// TIA Portal V17 export
// export: Created 2024-08-26T21:07:16.6253972Z, ExportSetting WithDefaults, DisplayName Totally Integrated Automation Portal, DisplayVersion V17 Update 7, DisplayName TIA Portal Openness, DisplayVersion V17 Update 7, DisplayName TIA Portal Version Control Interface, DisplayVersion V17, DisplayName SINAMICS Startdrive Advanced, DisplayVersion V17 SP2, DisplayName SINAMICS Startdrive G110M, G120, G120C, G120D, G120P, G115D, DisplayVersion V17 SP2, DisplayName SINAMICS Startdrive G130, G150, S120, S150, SINAMICS MV, S210, DisplayVersion V17 SP2, DisplayName STEP 7 Professional, DisplayVersion V17 Update 7, DisplayName STEP 7 Safety, DisplayVersion V17 Update 6, DisplayName WinCC Advanced / Unified PC, DisplayVersion V17 Update 7
DATA_BLOCK "torque"   // DB34
{ S7_Optimized_Access := 'TRUE' }
VERSION : 0.1
// stored: AutoNumber true, DBAccessibleFromOPCUA true, DBAccessibleFromWebserver true, IsOnlyStoredInLoadMemory false, IsRetainMemResEnabled false, IsWriteProtectedInAS false, MemoryReserve 100
   VAR
      ON : Bool := FALSE;
      SENSOR : Int := 0;
      TORQUE : Int := 0;
      TIMER1 { S7_SetPoint := 'True'} : TON_TIME;
      TIMER2 { S7_SetPoint := 'True'} : TON_TIME;
      TIMER3 { S7_SetPoint := 'True'} : TON_TIME;
      TIMER4 { S7_SetPoint := 'True'} : TON_TIME;
      TIMER5 { S7_SetPoint := 'True'} : TON_TIME;
      "1stInt" : Word := 16#0000;
      "2ndInt" : Word := 16#0000;
      "3rdInt" : Word := 16#0000;
      "4thInt" : Word := 16#0000;
      "5thInt" : Word := 16#0000;
      "1stDecimal" : Word := 16#0000;
      "2ndDecimal" : Word := 16#0000;
      "3rdDecimal" : Word := 16#0000;
      "4thDecimal" : Word := 16#0000;
      "5thDecimal" : Word := 16#0000;
      "1stFinalAngle" : Word := 16#0000;
      "2ndFinalAngle" : Word := 16#0000;
      "3rdFinalAngle" : Word := 16#0000;
      "4thFinalAngle" : Word := 16#0000;
      "5thFinalAngle" : Word := 16#0000;
      "ENTERO MANUAL" : Word := 16#0000;
      "DECIMAL MANUAL" : Word := 16#0000;
      "ANGULO FINAL MANUAL" : Word := 16#0000;
      TORNILLO : Int := 0;
      "1Ok" : Bool := FALSE;
      "2Ok" : Bool := FALSE;
      "3Ok" : Bool := FALSE;
      "4Ok" : Bool := FALSE;
      "1_OK_2" : Bool := FALSE;
      "2_OK_2" : Bool := FALSE;
      "3_OK_2" : Bool := FALSE;
      "4_OK_2" : Bool := FALSE;
      "5_OK_2" : Bool := FALSE;
      "5_OK" : Bool := FALSE;
      "ACTIVAR MANUAL" : Bool := FALSE;
      "CONFIG1 MANUAL" : Bool := FALSE;
      "CONFIG2 MANUAL" : Bool := FALSE;
      "CONFIG3 MANUAL" : Bool := FALSE;
      "CONFIG4 MANUAL" : Bool := FALSE;
      "CONFIG5 MANUAL" : Bool := FALSE;
      "REINICIAR PFJOB" : Bool := FALSE;
      PRESET1 : Int := 0;
      PRESET2 : Int := 0;
      PRESET3 : Int := 0;
      PRESET4 : Int := 0;
      PRESET5 : Int := 0;
      manual2 : Struct
         HABILITAR : Bool := TRUE;
         DESHABILITAR : Bool := FALSE;
         BORRAR : Bool := FALSE;
      END_STRUCT;
      BLOQUEO : Array[0..6] of Bool;
      manual : Struct
         activate : Bool := TRUE;
         deactivate : Bool := FALSE;
         erase : Bool := FALSE;
      END_STRUCT;
   END_VAR
   VAR RETAIN
      "P6000 TORQUE_1" : Array[0..15] of Int;
      p6000Torque : Array[0..15] of Int;
   END_VAR
   VAR
      nok2 : Array[0..1] of Bool;
      nok : Array[0..1] of Bool;
   END_VAR
BEGIN
   TIMER1.PT := T#0MS;
   TIMER1.IN := FALSE;
   TIMER2.PT := T#0MS;
   TIMER2.IN := FALSE;
   TIMER3.PT := T#0MS;
   TIMER3.IN := FALSE;
   TIMER4.PT := T#0MS;
   TIMER4.IN := FALSE;
   TIMER5.PT := T#0MS;
   TIMER5.IN := FALSE;
   BLOQUEO[0..6] := FALSE;
   "P6000 TORQUE_1"[0] := 1;
   "P6000 TORQUE_1"[1] := 2;
   "P6000 TORQUE_1"[2] := 3;
   "P6000 TORQUE_1"[3] := 1;
   "P6000 TORQUE_1"[4] := 2;
   "P6000 TORQUE_1"[5] := 3;
   "P6000 TORQUE_1"[6..15] := 0;
   p6000Torque[0] := 1;
   p6000Torque[1] := 2;
   p6000Torque[2] := 3;
   p6000Torque[3] := 1;
   p6000Torque[4] := 2;
   p6000Torque[5] := 3;
   p6000Torque[6..15] := 0;
   nok2[0..1] := FALSE;
   nok[0..1] := FALSE;
END_DATA_BLOCK
